(* IEC 61131-3 sources: PLCpilot/plc_programs, 4 files *)

(* ---- pump_alternation.st ---- *)
PROGRAM PumpAlternate
VAR
    PumpA         AT %QX0.0 : BOOL;
    PumpB         AT %QX0.1 : BOOL;
    Timer12H      : TON;
    ActivePump    : BOOL := FALSE;
END_VAR

Timer12H(IN := TRUE, PT := T#43200s);

IF Timer12H.Q THEN
    ActivePump := NOT ActivePump;
    Timer12H(IN := FALSE, PT := T#43200s);
    Timer12H(IN := TRUE, PT := T#43200s);
END_IF;

PumpA := NOT ActivePump;
PumpB := ActivePump;
END_PROGRAM

CONFIGURATION Config0
    RESOURCE Res0 ON PLC
        TASK MainTask(INTERVAL := T#100ms, PRIORITY := 1);
        PROGRAM PumpInst WITH MainTask : PumpAlternate;
    END_RESOURCE
END_CONFIGURATION

(* ---- sensor_drift_robotic_arm.st ---- *)
PROGRAM SensorDriftDetect
VAR
    ActualPos     AT %MW0 : INT;
    ExpectedPos   AT %MW1 : INT;
    DriftAlarm    AT %QX0.0 : BOOL;
    SafetyStop    AT %QX0.1 : BOOL;
    Drift         : INT;
END_VAR

VAR CONSTANT
    DRIFT_LIMIT : INT := 50;
END_VAR

Drift := ActualPos - ExpectedPos;
IF Drift < 0 THEN
    Drift := -Drift;
END_IF;

IF Drift > DRIFT_LIMIT THEN
    DriftAlarm := TRUE;
    SafetyStop := TRUE;
ELSE
    DriftAlarm := FALSE;
    SafetyStop := FALSE;
END_IF;
END_PROGRAM

CONFIGURATION Config0
    RESOURCE Res0 ON PLC
        TASK MainTask(INTERVAL := T#100ms, PRIORITY := 1);
        PROGRAM DriftInst WITH MainTask : SensorDriftDetect;
    END_RESOURCE
END_CONFIGURATION

(* ---- temp_fan_control.st ---- *)
PROGRAM TempControl
VAR
    TempSensor AT %MW0 : INT;
    Fan        AT %QX0.0 : BOOL;
    Alarm      AT %QX0.1 : BOOL;
END_VAR

VAR CONSTANT
    HIGH_LIMIT : INT := 75;
    LOW_LIMIT  : INT := 70;
END_VAR

IF TempSensor >= HIGH_LIMIT THEN
    Fan := TRUE;
    Alarm := TRUE;
ELSIF TempSensor <= LOW_LIMIT THEN
    Fan := FALSE;
    Alarm := FALSE;
END_IF;
END_PROGRAM

CONFIGURATION Config0
    RESOURCE Res0 ON PLC
        TASK MainTask(INTERVAL := T#100ms, PRIORITY := 1);
        PROGRAM TempInst WITH MainTask : TempControl;
    END_RESOURCE
END_CONFIGURATION

(* ---- watchdog_press.st ---- *)
PROGRAM WatchdogPress
VAR
    SensorPulse   AT %IX0.0 : BOOL;
    MachineRun    AT %QX0.0 : BOOL;
    WatchdogTimer : TON;
    LastPulse     : BOOL;
END_VAR

WatchdogTimer(IN := NOT SensorPulse, PT := T#10s);

IF WatchdogTimer.Q THEN
    MachineRun := FALSE;
END_IF;

IF SensorPulse AND NOT LastPulse THEN
    MachineRun := TRUE;
    WatchdogTimer(IN := FALSE, PT := T#10s);
END_IF;

LastPulse := SensorPulse;
END_PROGRAM

CONFIGURATION Config0
    RESOURCE Res0 ON PLC
        TASK MainTask(INTERVAL := T#100ms, PRIORITY := 1);
        PROGRAM WatchdogInst WITH MainTask : WatchdogPress;
    END_RESOURCE
END_CONFIGURATION
